FUNCTION_BLOCK T_NotificationHandler IMPLEMENTS I_NotificationHandler
VAR
    _Args            : T_Stream(StreamLength := 4);
    _IsRaised        : BOOL;
    _InvocationCount : DINT;
END_VAR

PROPERTY Args : I_StreamReader
GET
Args := _Args;
END_GET
END_PROPERTY

METHOD Handled
VAR_INPUT
END_VAR
_IsRaised := FALSE;
_InvocationCount := 0;
END_METHOD

PROPERTY InvocationCount : DINT
GET
InvocationCount := _InvocationCount;
END_GET
END_PROPERTY

METHOD IsRaised : BOOL
VAR_INPUT
END_VAR
IsRaised := _IsRaised;
END_METHOD

METHOD OnNotificationReceived
VAR_INPUT
    NotificationId   : UDINT;
    NotificationName : Tc2_System.T_MaxString;
    Args             : I_StreamReader;
END_VAR
VAR
    i          : UDINT;
    ByteToCopy : BYTE;
END_VAR
IF Args.ByteCount > 0 THEN // has event arguments..
    _Args.CopyFromStreamReader(Args);
END_IF

_Args.Seek(0);

_IsRaised          := TRUE;
// keep track of how many times it has been raised so we can count number of notifications between being handled
_InvocationCount := _InvocationCount + 1;
END_METHOD

END_FUNCTION_BLOCK

(* stored: Version 1.1.0.1, ProductVersion 3.1.4024.6
   POU T_NotificationHandler: Id {607f5e14-d01e-4493-979d-0fc6e8f214bb}, SpecialFunc None
   Folder Methods: Id {50523a27-f4f0-421d-b359-9106ca91093f}
   Folder Properties: Id {fa028168-01fb-46c8-9542-d1715323a920}
   Property Args: Id {91257052-647a-4693-b950-dbd5f4670b44}
   Get Get: Id {53b1bc30-dc6e-49ed-9d6e-3cc453a91aed}
   Method Handled: Id {66e16aac-78b8-424e-a9ed-840351f5e3bd}
   Property InvocationCount: Id {5bd3cb2d-5961-41b2-9319-18b3e8af94e2}
   Get Get: Id {fb9ecc7c-8d9e-4665-b605-3ba3bba5a0d2}
   Method IsRaised: Id {fae0f454-b76e-425b-b849-6b812d700aa5}
   Method OnNotificationReceived: Id {8767452b-6194-4156-b4a1-080cf2d33e36} *)
